// TIA Portal V19 export
DATA_BLOCK "LAcycCom_RequestBuffer"   // DB3348
TITLE = LAcycCom_RequestBuffer
{ S7_Optimized_Access := 'TRUE' }
AUTHOR : APC_ERLF
FAMILY : AcycCom
VERSION : 1.2
// Support: tech.team.motioncontrol@siemens.com 
// Fax: +49 (0) 9131/98-1297
// stored: InstanceOfName LAcycCom_typeRequestBuffer, InstanceOfType UDT
"LAcycCom_typeRequestBuffer"
   // VAR
   //    header { ExternalAccessible := 'False'; ExternalVisible := 'False'; ExternalWritable := 'False'; S7_SetPoint := 'True'} : "LAcycCom_typeRequestBufferHeader";
   //    elements { ExternalAccessible := 'False'; ExternalVisible := 'False'; ExternalWritable := 'False'; S7_SetPoint := 'True'} : Array[0.."LACYCCOM_BUFFER_ELEMENTS_UPPER_LIM"] of "LAcycCom_typeRequestBufferElement";
   // END_VAR
BEGIN
END_DATA_BLOCK
